// TIA Portal project "FactoryIO_Template_S7-1200_V16_V16" (V16)
// Vorlageprojekt für das Buch mit Zielsystem S7-1200

(* hardware
DEVICE "S7-1200-Station_1"  S7-1200 Station
   slot 0: "Baugruppenträger_0"  Rack  V1.0
   slot 1: "PLC_1"  CPU 1211C DC/DC/DC  6ES7 211-1AE40-0XB0  V4.1
*)

// ===== PLC "PLC_1"  CPU 1211C DC/DC/DC =====

VAR_GLOBAL   // PLC tag table "Standard-Variablentabelle"
   "AT ENTRY" AT %I0.0 : Bool;
   "AT LOAD" AT %I0.1 : Bool;
   "AT LEFT" AT %I0.2 : Bool;
   "AT MIDDLE" AT %I0.3 : Bool;
   "AT RIGHT" AT %I0.4 : Bool;
   "AT UNLOAD" AT %I0.5 : Bool;
   "AT EXIT" AT %I0.6 : Bool;
   "MOVING X" AT %I0.7 : Bool;
   "MOVING Z" AT %I1.0 : Bool;
   "START" AT %I1.1 : Bool;
   "RESET" AT %I1.2 : Bool;
   "STOP" AT %I1.3 : Bool;
   "EMERGENCY STOP" AT %I1.4 : Bool;
   "AUTO" AT %I1.5 : Bool;
   "ENTRY CONVEYOR" AT %Q0.0 : Bool;
   "LOAD CONVEYOR" AT %Q0.1 : Bool;
   "FORKS LEFT" AT %Q0.2 : Bool;
   "FORKS RIGHT" AT %Q0.3 : Bool;
   "LIFT" AT %Q0.4 : Bool;
   "UNLOAD CONVEYOR" AT %Q0.5 : Bool;
   "EXIT CONVEYOR" AT %Q0.6 : Bool;
   "START LIGHT" AT %Q0.7 : Bool;
   "RESET LIGHT" AT %Q1.0 : Bool;
   "STOP LIGHT" AT %Q1.1 : Bool;
   "TARGET POSITION" AT %QD30 : DInt;
   "STATE1" AT %M0.0 : Bool;
   "STATE2" AT %M0.1 : Bool;
   "STATE3" AT %M0.2 : Bool;
   "STATE4" AT %M0.3 : Bool;
   "STATE5" AT %M0.4 : Bool;
   "STATE6" AT %M0.5 : Bool;
   "STATE7" AT %M0.6 : Bool;
   "STATE8" AT %M0.7 : Bool;
   "STATE9" AT %M1.0 : Bool;
   "STATE10" AT %M1.1 : Bool;
   "Tag_1" AT %MD2 : DInt;
   "Tag_2" AT %MD6 : DInt;
   "M1" AT %M1.2 : Bool;
   "M2" AT %M1.3 : Bool;
   "M3" AT %M1.4 : Bool;
   "M4" AT %M1.5 : Bool;
   "M5" AT %M1.6 : Bool;
   "M6" AT %M1.7 : Bool;
   "M7" AT %M10.0 : Bool;
END_VAR

FUNCTION "START_STOP" : Void   // FC1, LAD
{ S7_Optimized_Access := 'TRUE' }
VERSION : 0.1
BEGIN

REGION Network 1
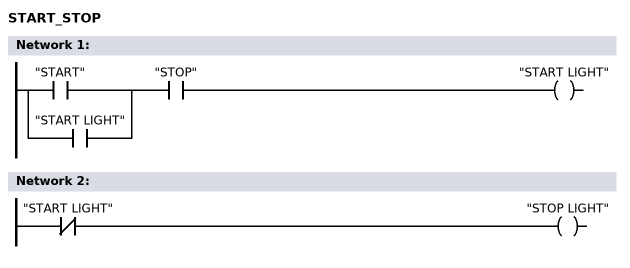
   RUNG wire#powerrail
      Contact( "START" )
      wire#w1
      Contact( "STOP" )
      Coil( "START LIGHT" )
   END_RUNG
   RUNG wire#powerrail
      Contact( "START LIGHT" )
   END_RUNG wire#w1
   // the same network as SCL:
   "START LIGHT" := ("START" OR "START LIGHT") AND "STOP";
END_REGION

REGION Network 2
   RUNG wire#powerrail
      I_Contact( "START LIGHT" )
      Coil( "STOP LIGHT" )
   END_RUNG
   // the same network as SCL:
   "STOP LIGHT" := NOT "START LIGHT";
END_REGION
END_FUNCTION

FUNCTION "ACUTATOR" : Void   // FC2, LAD
{ S7_Optimized_Access := 'TRUE' }
VERSION : 0.1
   VAR_TEMP   // added for the SCL form of the ladder/FBD networks
      _w1 : Bool;
   END_VAR
BEGIN

REGION Network 1
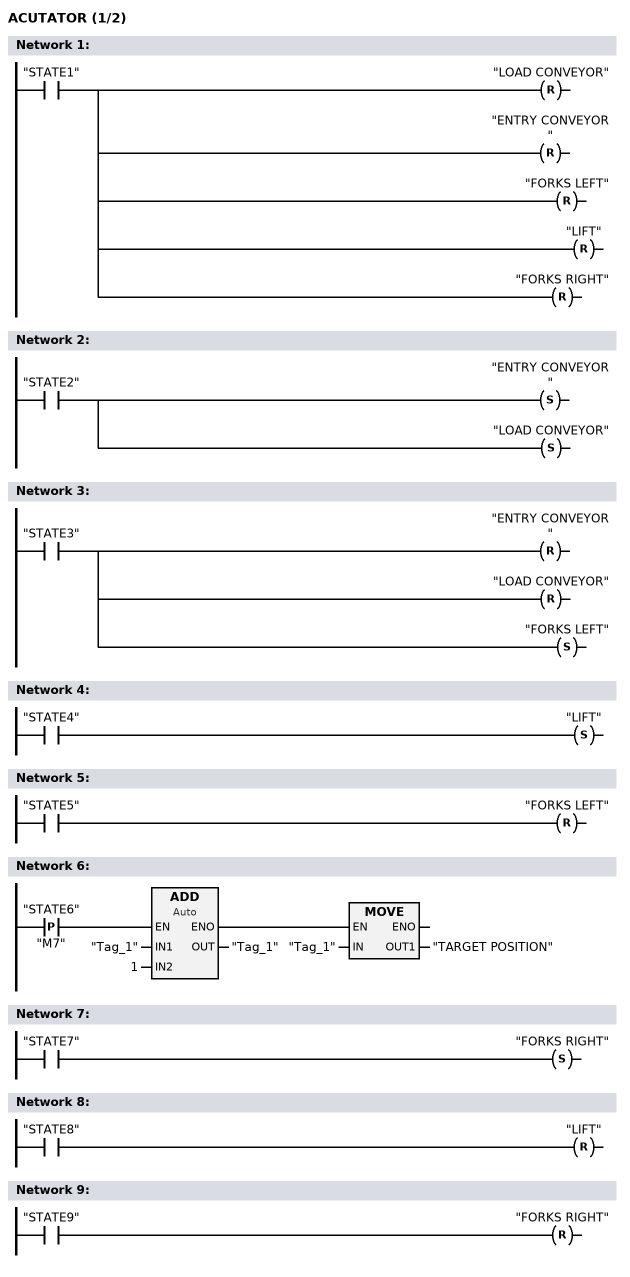
   RUNG wire#powerrail
      Contact( "STATE1" )
      wire#w1
      R_Coil( "LOAD CONVEYOR" )
   END_RUNG
   RUNG wire#w1
      R_Coil( "ENTRY CONVEYOR" )
   END_RUNG
   RUNG wire#w1
      R_Coil( "FORKS LEFT" )
   END_RUNG
   RUNG wire#w1
      R_Coil( "LIFT" )
   END_RUNG
   RUNG wire#w1
      R_Coil( "FORKS RIGHT" )
   END_RUNG
   // the same network as SCL:
   IF "STATE1" THEN
       "LOAD CONVEYOR" := FALSE;
       "ENTRY CONVEYOR" := FALSE;
       "FORKS LEFT" := FALSE;
       "LIFT" := FALSE;
       "FORKS RIGHT" := FALSE;
   END_IF;
END_REGION

REGION Network 2
   RUNG wire#powerrail
      Contact( "STATE2" )
      wire#w1
      S_Coil( "ENTRY CONVEYOR" )
   END_RUNG
   RUNG wire#w1
      S_Coil( "LOAD CONVEYOR" )
   END_RUNG
   // the same network as SCL:
   IF "STATE2" THEN
       "ENTRY CONVEYOR" := TRUE;
       "LOAD CONVEYOR" := TRUE;
   END_IF;
END_REGION

REGION Network 3
   RUNG wire#powerrail
      Contact( "STATE3" )
      wire#w1
      R_Coil( "ENTRY CONVEYOR" )
   END_RUNG
   RUNG wire#w1
      R_Coil( "LOAD CONVEYOR" )
   END_RUNG
   RUNG wire#w1
      S_Coil( "FORKS LEFT" )
   END_RUNG
   // the same network as SCL:
   IF "STATE3" THEN
       "ENTRY CONVEYOR" := FALSE;
       "LOAD CONVEYOR" := FALSE;
       "FORKS LEFT" := TRUE;
   END_IF;
END_REGION

REGION Network 4
   RUNG wire#powerrail
      Contact( "STATE4" )
      S_Coil( "LIFT" )
   END_RUNG
   // the same network as SCL:
   IF "STATE4" THEN "LIFT" := TRUE; END_IF;
END_REGION

REGION Network 5
   RUNG wire#powerrail
      Contact( "STATE5" )
      R_Coil( "FORKS LEFT" )
   END_RUNG
   // the same network as SCL:
   IF "STATE5" THEN "FORKS LEFT" := FALSE; END_IF;
END_REGION

REGION Network 6
   RUNG wire#powerrail
      P_Contact(operand := "STATE6", bit := "M7")
      Add(in1 := "Tag_1", in2 := 1, out => "Tag_1")
      Move(in := "Tag_1", out1 => "TARGET POSITION")
   END_RUNG
   // the same network as SCL:
   #_w1 := "STATE6" AND NOT "M7";   // rising edge of "STATE6"
   "M7" := "STATE6";
   IF #_w1 THEN
       "Tag_1" := "Tag_1" + 1;
       "TARGET POSITION" := "Tag_1";
   END_IF;
END_REGION

REGION Network 7
   RUNG wire#powerrail
      Contact( "STATE7" )
      S_Coil( "FORKS RIGHT" )
   END_RUNG
   // the same network as SCL:
   IF "STATE7" THEN "FORKS RIGHT" := TRUE; END_IF;
END_REGION

REGION Network 8
   RUNG wire#powerrail
      Contact( "STATE8" )
      R_Coil( "LIFT" )
   END_RUNG
   // the same network as SCL:
   IF "STATE8" THEN "LIFT" := FALSE; END_IF;
END_REGION

REGION Network 9
   RUNG wire#powerrail
      Contact( "STATE9" )
      R_Coil( "FORKS RIGHT" )
   END_RUNG
   // the same network as SCL:
   IF "STATE9" THEN "FORKS RIGHT" := FALSE; END_IF;
END_REGION

REGION Network 10
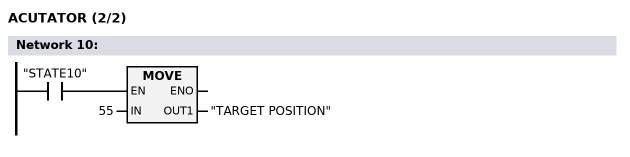
   RUNG wire#powerrail
      Contact( "STATE10" )
      Move(in := 55, out1 => "TARGET POSITION")
   END_RUNG
   // the same network as SCL:
   IF "STATE10" THEN "TARGET POSITION" := 55; END_IF;
END_REGION
END_FUNCTION

FUNCTION "STATES" : Void   // FC3, LAD
{ S7_Optimized_Access := 'TRUE' }
VERSION : 0.1
   VAR_TEMP   // added for the SCL form of the ladder/FBD networks
      _w1 : Bool;
      _w2 : Bool;
      _w3 : Bool;
      _w4 : Bool;
   END_VAR
BEGIN

REGION Network 1
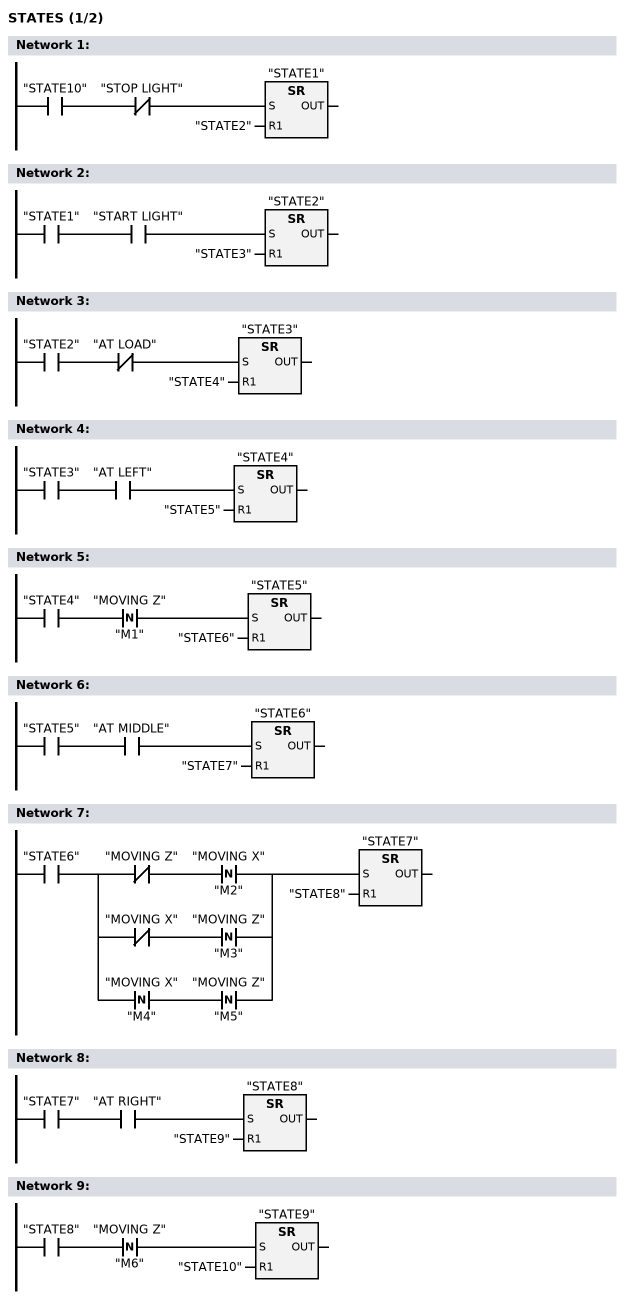
   RUNG wire#powerrail
      Contact( "STATE10" )
      I_Contact( "STOP LIGHT" )
      S_SR(operand := "STATE1", r1 := "STATE2")
   END_RUNG
   // the same network as SCL:
   IF "STATE10" AND NOT "STOP LIGHT" THEN
       "STATE1" := TRUE;   // SR flip-flop
   END_IF;
   IF "STATE2" THEN "STATE1" := FALSE; END_IF;
END_REGION

REGION Network 2
   RUNG wire#powerrail
      Contact( "STATE1" )
      Contact( "START LIGHT" )
      S_SR(operand := "STATE2", r1 := "STATE3")
   END_RUNG
   // the same network as SCL:
   IF "STATE1" AND "START LIGHT" THEN
       "STATE2" := TRUE;   // SR flip-flop
   END_IF;
   IF "STATE3" THEN "STATE2" := FALSE; END_IF;
END_REGION

REGION Network 3
   RUNG wire#powerrail
      Contact( "STATE2" )
      I_Contact( "AT LOAD" )
      S_SR(operand := "STATE3", r1 := "STATE4")
   END_RUNG
   // the same network as SCL:
   IF "STATE2" AND NOT "AT LOAD" THEN
       "STATE3" := TRUE;   // SR flip-flop
   END_IF;
   IF "STATE4" THEN "STATE3" := FALSE; END_IF;
END_REGION

REGION Network 4
   RUNG wire#powerrail
      Contact( "STATE3" )
      Contact( "AT LEFT" )
      S_SR(operand := "STATE4", r1 := "STATE5")
   END_RUNG
   // the same network as SCL:
   IF "STATE3" AND "AT LEFT" THEN
       "STATE4" := TRUE;   // SR flip-flop
   END_IF;
   IF "STATE5" THEN "STATE4" := FALSE; END_IF;
END_REGION

REGION Network 5
   RUNG wire#powerrail
      Contact( "STATE4" )
      N_Contact(operand := "MOVING Z", bit := "M1")
      S_SR(operand := "STATE5", r1 := "STATE6")
   END_RUNG
   // the same network as SCL:
   #_w1 := "STATE4" AND NOT "MOVING Z" AND "M1";   // falling edge of "MOVING Z"
   "M1" := "MOVING Z";
   IF #_w1 THEN
       "STATE5" := TRUE;   // SR flip-flop
   END_IF;
   IF "STATE6" THEN "STATE5" := FALSE; END_IF;
END_REGION

REGION Network 6
   RUNG wire#powerrail
      Contact( "STATE5" )
      Contact( "AT MIDDLE" )
      S_SR(operand := "STATE6", r1 := "STATE7")
   END_RUNG
   // the same network as SCL:
   IF "STATE5" AND "AT MIDDLE" THEN
       "STATE6" := TRUE;   // SR flip-flop
   END_IF;
   IF "STATE7" THEN "STATE6" := FALSE; END_IF;
END_REGION

REGION Network 7
   RUNG wire#powerrail
      Contact( "STATE6" )
      wire#w1
      I_Contact( "MOVING Z" )
      N_Contact(operand := "MOVING X", bit := "M2")
      wire#w2
      S_SR(operand := "STATE7", r1 := "STATE8")
   END_RUNG
   RUNG wire#w1
      I_Contact( "MOVING X" )
      N_Contact(operand := "MOVING Z", bit := "M3")
   END_RUNG wire#w2
   RUNG wire#w1
      N_Contact(operand := "MOVING X", bit := "M4")
      N_Contact(operand := "MOVING Z", bit := "M5")
   END_RUNG wire#w2
   // the same network as SCL:
   #_w1 := "STATE6" AND NOT "MOVING Z" AND NOT "MOVING X" AND "M2";   // falling edge of "MOVING X"
   "M2" := "MOVING X";
   #_w2 := "STATE6" AND NOT "MOVING X" AND NOT "MOVING Z" AND "M3";   // falling edge of "MOVING Z"
   "M3" := "MOVING Z";
   #_w3 := "STATE6" AND NOT "MOVING X" AND "M4";   // falling edge of "MOVING X"
   "M4" := "MOVING X";
   #_w4 := #_w3 AND NOT "MOVING Z" AND "M5";   // falling edge of "MOVING Z"
   "M5" := "MOVING Z";
   IF #_w1 OR #_w2 OR #_w4 THEN
       "STATE7" := TRUE;   // SR flip-flop
   END_IF;
   IF "STATE8" THEN "STATE7" := FALSE; END_IF;
END_REGION

REGION Network 8
   RUNG wire#powerrail
      Contact( "STATE7" )
      Contact( "AT RIGHT" )
      S_SR(operand := "STATE8", r1 := "STATE9")
   END_RUNG
   // the same network as SCL:
   IF "STATE7" AND "AT RIGHT" THEN
       "STATE8" := TRUE;   // SR flip-flop
   END_IF;
   IF "STATE9" THEN "STATE8" := FALSE; END_IF;
END_REGION

REGION Network 9
   RUNG wire#powerrail
      Contact( "STATE8" )
      N_Contact(operand := "MOVING Z", bit := "M6")
      S_SR(operand := "STATE9", r1 := "STATE10")
   END_RUNG
   // the same network as SCL:
   #_w1 := "STATE8" AND NOT "MOVING Z" AND "M6";   // falling edge of "MOVING Z"
   "M6" := "MOVING Z";
   IF #_w1 THEN
       "STATE9" := TRUE;   // SR flip-flop
   END_IF;
   IF "STATE10" THEN "STATE9" := FALSE; END_IF;
END_REGION

REGION Network 10
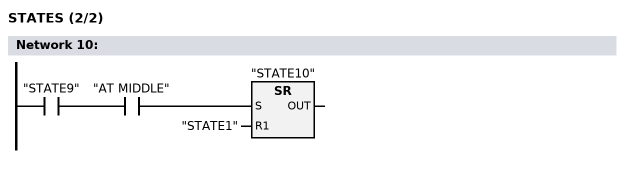
   RUNG wire#powerrail
      Contact( "STATE9" )
      Contact( "AT MIDDLE" )
      S_SR(operand := "STATE10", r1 := "STATE1")
   END_RUNG
   // the same network as SCL:
   IF "STATE9" AND "AT MIDDLE" THEN
       "STATE10" := TRUE;   // SR flip-flop
   END_IF;
   IF "STATE1" THEN "STATE10" := FALSE; END_IF;
END_REGION
END_FUNCTION

FUNCTION "MHJ-PLC-Lab-Function-S71200" : Void   // FC9000, SCL
{ S7_Optimized_Access := 'TRUE' }
VERSION : 0.1
   VAR_TEMP
      rdTimeReturn : Int;
      outputTime : DTL;
      SyncVal : Byte;
      forVal : Int;
      forVal_2 : Int;
      Value : Byte;
   END_VAR
   VAR CONSTANT
      CompVal : Byte := 16#34;
      Value_01 : Byte := 16#11;
      Value_01_DW : DWord := 16#A165_D992;
      Value_02_DW : DWord := 16#58BE_4401;
   END_VAR
BEGIN

   #Value:=PEEK(area := 16#82,
        dbNumber := 0,
        byteOffset := 511);
   #Value := #Value + 1;

   POKE(area := 16#82,
        dbNumber := 0,
        byteOffset := 511,
        value := #Value);

   POKE(area:=16#81,
        dbNumber:=0,
        byteOffset:=1016,
        value:=#Value_01_DW);
   POKE(area := 16#81,
        dbNumber := 0,
        byteOffset := 1020,
        value := #Value_02_DW);

   POKE(area := 16#81,
        dbNumber := 0,
        byteOffset := 511,
        value := B#16#00);

   FOR #forVal := 0 TO 120 DO
       FOR #forVal_2:=0 TO 10 DO
           #rdTimeReturn:=RD_SYS_T(#outputTime);
           #rdTimeReturn := WR_SYS_T(#outputTime);
           #rdTimeReturn := RD_SYS_T(#outputTime);
           #rdTimeReturn := WR_SYS_T(#outputTime);
       END_FOR;
       #SyncVal:= PEEK(area := 16#81,
                      dbNumber := 0,
                      byteOffset := 511);
       IF #SyncVal = #CompVal THEN
          GOTO M_1;
       END_IF;
   END_FOR;
   RETURN;

   M_1:
   POKE(area := 16#81,
        dbNumber := 0,
        byteOffset := 511,
        value := B#16#0);
END_FUNCTION

ORGANIZATION_BLOCK "Main"   // OB1, LAD, ProgramCycle
TITLE = "Main Program Sweep (Cycle)"
{ S7_Optimized_Access := 'TRUE' }
VERSION : 0.1
   VAR_INPUT
      Initial_Call : Bool;   // Initial call of this OB
      Remanence : Bool;   // =True, if remanent data are available
   END_VAR
BEGIN

REGION Network 1: Konnektierungsbaustein für PLC-Lab
   // Im Netzwerk 1 wird der Konnektierungsbaustein für PLC-Lab aufgerufen.
   // Dieser Aufruf darf nicht entfernt werden!
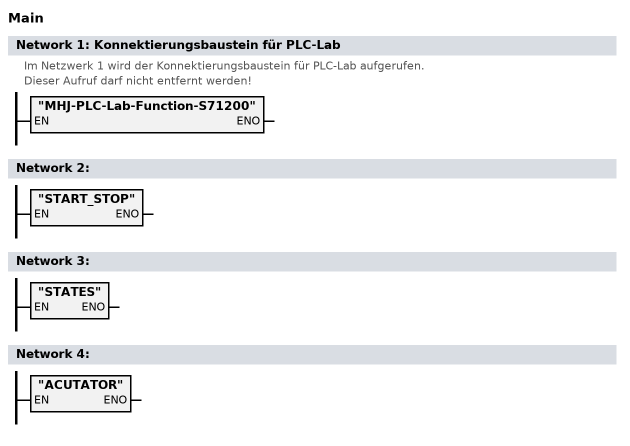
   RUNG wire#powerrail
      "MHJ-PLC-Lab-Function-S71200"()
   END_RUNG
   // the same network as SCL:
   "MHJ-PLC-Lab-Function-S71200"();
END_REGION

REGION Network 2
   RUNG wire#powerrail
      "START_STOP"()
   END_RUNG
   // the same network as SCL:
   "START_STOP"();
END_REGION

REGION Network 3
   RUNG wire#powerrail
      "STATES"()
   END_RUNG
   // the same network as SCL:
   "STATES"();
END_REGION

REGION Network 4
   RUNG wire#powerrail
      "ACUTATOR"()
   END_RUNG
   // the same network as SCL:
   "ACUTATOR"();
END_REGION
END_ORGANIZATION_BLOCK

ORGANIZATION_BLOCK "Startup"   // OB100, LAD, Startup
TITLE = "Complete Restart"
{ S7_Optimized_Access := 'TRUE' }
VERSION : 0.1
   VAR_INPUT
      LostRetentive : Bool;   // True if retentive data are lost
      LostRTC : Bool;   // True if date and time are lost
   END_VAR
BEGIN

REGION Network 1
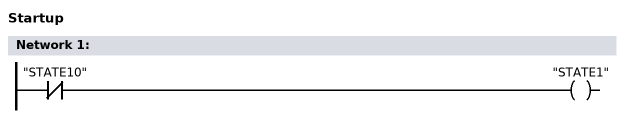
   RUNG wire#powerrail
      I_Contact( "STATE10" )
      Coil( "STATE1" )
   END_RUNG
   // the same network as SCL:
   "STATE1" := NOT "STATE10";
END_REGION
END_ORGANIZATION_BLOCK